// TIA Portal V19 export
TYPE "LEXCHANGETRAY_typeSr1000ProfinetTelegram_handshakAndGeneralErrorStatusBits"
// stored: Access Published
   STRUCT
      statusByte : Byte;
      error : Bool;
      resultDataAvailable : Bool;
      resultDataStrobe : Bool;
      bufferOverflowError : Bool;
      generalError : Bool;
   END_STRUCT;
END_TYPE
